(* IEC 61131-3 sources: Daniele1996.github.io/AUTOMATION_AND_SOFTWARE_DESIGN_PATTERN/AUTOMATION_STUDIO/Task2/Logical/MachineProgram, 3 files *)

(* ---- Types.typ ---- *)
TYPE
	Machine_States: (
					Machine_ready_to_be_initialized,
					Machine_initializing,
					Machine_ready_to_run,
					Conveyor_Enabling,
					Cutter_Enabling,
					Machine_on_phase_stopping);
END_TYPE

(* ---- Main.st ---- *)
PROGRAM _CYCLIC
	(* Insert code here *)
	CASE state OF

		Machine_ready_to_be_initialized:
			IF Machine_Handler.Initialize THEN
				Conveyor_Handler.Initialize := TRUE;
				Cutter_Handler.Initialize := TRUE;

				state := Machine_initializing;
			END_IF;

		Machine_initializing:
			IF NOT Conveyor_Handler.Initialize AND NOT Cutter_Handler.Initialize THEN
				Machine_Handler.Initialize := FALSE;

				state := Machine_ready_to_run;
			END_IF;

		Machine_ready_to_run:
			IF Machine_Handler.Run THEN
				Conveyor_Handler.Enable := TRUE;

				state := Conveyor_Enabling;
			END_IF;

		Conveyor_Enabling:
			IF Machine_Handler.On_Phase_Stop THEN
				Conveyor_Handler.On_Phase_Stop := TRUE;
				Cutter_Handler.On_Phase_Stop := TRUE;

				state := Machine_on_phase_stopping;

			ELSIF NOT Conveyor_Handler.Enable AND Trigger_logical THEN
				Cutter_Handler.Enable := TRUE;

				state := Cutter_Enabling;
			END_IF;

		Cutter_Enabling:
			IF NOT Cutter_Handler.Enable THEN

				state := Conveyor_Enabling;
			END_IF;

		Machine_on_phase_stopping:
			IF NOT Machine_Handler.On_Phase_Stop THEN
				Conveyor_Handler.On_Phase_Stop := FALSE;
				Cutter_Handler.On_Phase_Stop := FALSE;

				state := Machine_ready_to_run;
			END_IF;
	END_CASE;

END_PROGRAM

PROGRAM _EXIT
	(* Insert code here *)

END_PROGRAM

(* ---- Variables.var ---- *)
VAR
	state: Machine_States := Machine_ready_to_be_initialized;
END_VAR
